SYSTEM ServerTest
  APPLICATION ServerTestApp
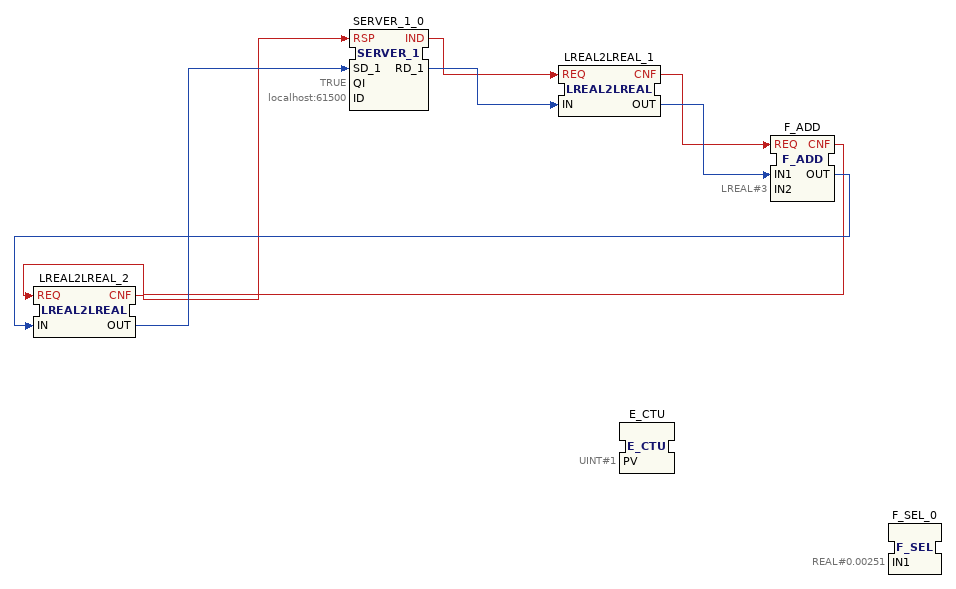
    FBS
      F_ADD : F_ADD(IN2 := LREAL#3);
      SERVER_1_0 : SERVER_1(QI := TRUE, ID := localhost:61500);
      LREAL2LREAL_1 : LREAL2LREAL;
      LREAL2LREAL_2 : LREAL2LREAL;
      E_CTU : E_CTU(PV := UINT#1);
      F_SEL_0 : F_SEL(IN1 := REAL#0.00251);
    END_FBS
    EVENT_CONNECTIONS
      SERVER_1_0.IND TO LREAL2LREAL_1.REQ;
      LREAL2LREAL_1.CNF TO F_ADD.REQ;
      F_ADD.CNF TO LREAL2LREAL_2.REQ;
      LREAL2LREAL_2.CNF TO SERVER_1_0.RSP;
    END_CONNECTIONS
    DATA_CONNECTIONS
      LREAL2LREAL_1.OUT TO F_ADD.IN1;
      SERVER_1_0.RD_1 TO LREAL2LREAL_1.IN;
      F_ADD.OUT TO LREAL2LREAL_2.IN;
      LREAL2LREAL_2.OUT TO SERVER_1_0.SD_1;
    END_CONNECTIONS
  END_APPLICATION
  APPLICATION ServerTestApp2
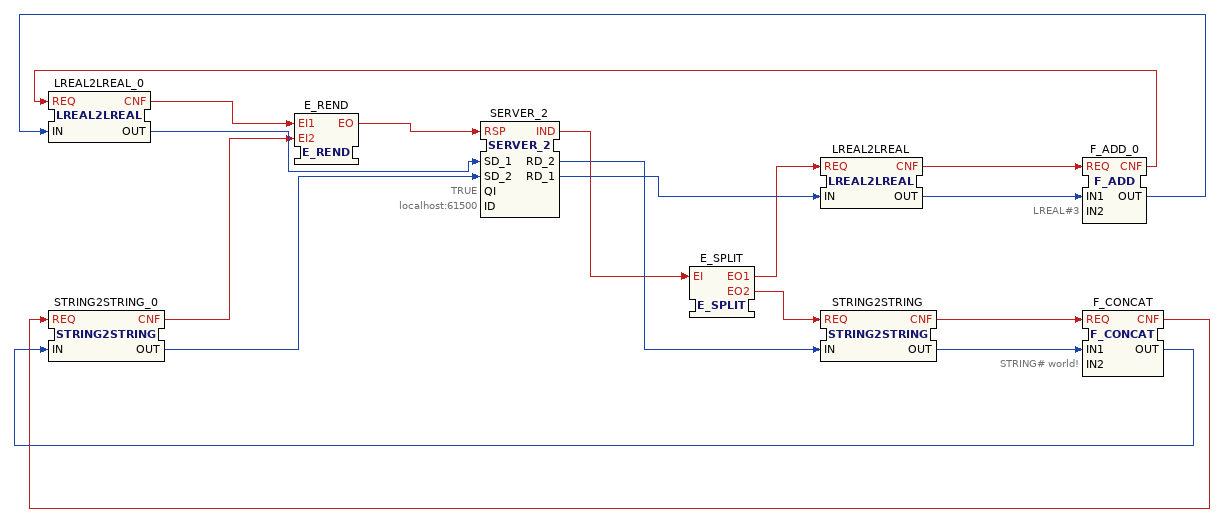
    FBS
      F_ADD_0 : F_ADD(IN2 := LREAL#3);
      F_CONCAT : F_CONCAT(IN2 := STRING# world!);
      SERVER_2 : SERVER_2(QI := TRUE, ID := localhost:61500);
      STRING2STRING : STRING2STRING;
      LREAL2LREAL : LREAL2LREAL;
      E_SPLIT : E_SPLIT;
      E_REND : E_REND;
      STRING2STRING_0 : STRING2STRING;
      LREAL2LREAL_0 : LREAL2LREAL;
    END_FBS
    EVENT_CONNECTIONS
      SERVER_2.IND TO E_SPLIT.EI;
      E_SPLIT.EO1 TO LREAL2LREAL.REQ;
      E_SPLIT.EO2 TO STRING2STRING.REQ;
      LREAL2LREAL.CNF TO F_ADD_0.REQ;
      STRING2STRING.CNF TO F_CONCAT.REQ;
      F_ADD_0.CNF TO LREAL2LREAL_0.REQ;
      F_CONCAT.CNF TO STRING2STRING_0.REQ;
      LREAL2LREAL_0.CNF TO E_REND.EI1;
      STRING2STRING_0.CNF TO E_REND.EI2;
      E_REND.EO TO SERVER_2.RSP;
    END_CONNECTIONS
    DATA_CONNECTIONS
      SERVER_2.RD_2 TO STRING2STRING.IN;
      STRING2STRING.OUT TO F_CONCAT.IN1;
      SERVER_2.RD_1 TO LREAL2LREAL.IN;
      LREAL2LREAL.OUT TO F_ADD_0.IN1;
      F_ADD_0.OUT TO LREAL2LREAL_0.IN;
      F_CONCAT.OUT TO STRING2STRING_0.IN;
      LREAL2LREAL_0.OUT TO SERVER_2.SD_1;
      STRING2STRING_0.OUT TO SERVER_2.SD_2;
    END_CONNECTIONS
  END_APPLICATION
  APPLICATION ServerTestApp3
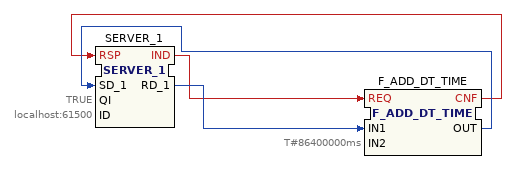
    FBS
      SERVER_1 : SERVER_1(QI := TRUE, ID := localhost:61500);
      F_ADD_DT_TIME : F_ADD_DT_TIME(IN2 := T#86400000ms);
    END_FBS
    EVENT_CONNECTIONS
      SERVER_1.IND TO F_ADD_DT_TIME.REQ;
      F_ADD_DT_TIME.CNF TO SERVER_1.RSP;
    END_CONNECTIONS
    DATA_CONNECTIONS
      SERVER_1.RD_1 TO F_ADD_DT_TIME.IN1;
      F_ADD_DT_TIME.OUT TO SERVER_1.SD_1;
    END_CONNECTIONS
  END_APPLICATION
  APPLICATION ServerTestApp4
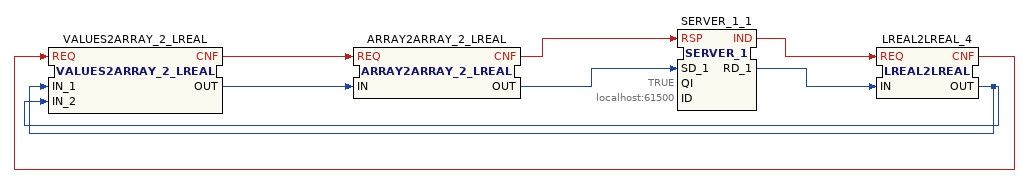
    FBS
      VALUES2ARRAY_2_LREAL : VALUES2ARRAY_2_LREAL;
      SERVER_1_1 : SERVER_1(QI := TRUE, ID := localhost:61500);
      ARRAY2ARRAY_2_LREAL : ARRAY2ARRAY_2_LREAL;
      LREAL2LREAL_4 : LREAL2LREAL;
    END_FBS
    EVENT_CONNECTIONS
      VALUES2ARRAY_2_LREAL.CNF TO ARRAY2ARRAY_2_LREAL.REQ;
      ARRAY2ARRAY_2_LREAL.CNF TO SERVER_1_1.RSP;
      SERVER_1_1.IND TO LREAL2LREAL_4.REQ;
      LREAL2LREAL_4.CNF TO VALUES2ARRAY_2_LREAL.REQ;
    END_CONNECTIONS
    DATA_CONNECTIONS
      VALUES2ARRAY_2_LREAL.OUT TO ARRAY2ARRAY_2_LREAL.IN;
      SERVER_1_1.RD_1 TO LREAL2LREAL_4.IN;
      LREAL2LREAL_4.OUT TO VALUES2ARRAY_2_LREAL.IN_1;
      LREAL2LREAL_4.OUT TO VALUES2ARRAY_2_LREAL.IN_2;
      ARRAY2ARRAY_2_LREAL.OUT TO SERVER_1_1.SD_1;
    END_CONNECTIONS
  END_APPLICATION
  APPLICATION ServerTest5
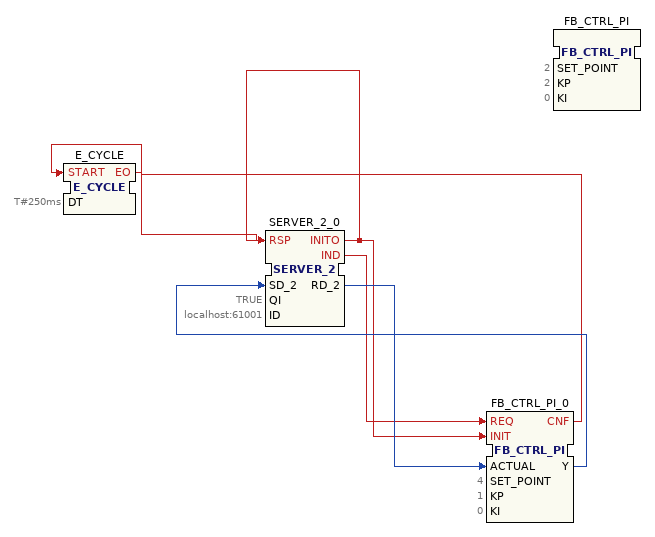
    FBS
      SERVER_2_0 : SERVER_2(QI := TRUE, ID := localhost:61001);
      FB_CTRL_PI : FB_CTRL_PI(SET_POINT := 2, KP := 2, KI := 0);
      FB_CTRL_PI_0 : FB_CTRL_PI(SET_POINT := 4, KP := 1, KI := 0);
      E_CYCLE : E_CYCLE(DT := T#250ms);
    END_FBS
    EVENT_CONNECTIONS
      SERVER_2_0.INITO TO SERVER_2_0.RSP;
      SERVER_2_0.IND TO FB_CTRL_PI_0.REQ;
      SERVER_2_0.INITO TO FB_CTRL_PI_0.INIT;
      FB_CTRL_PI_0.CNF TO E_CYCLE.START;
      E_CYCLE.EO TO SERVER_2_0.RSP;
    END_CONNECTIONS
    DATA_CONNECTIONS
      SERVER_2_0.RD_2 TO FB_CTRL_PI_0.ACTUAL;
      FB_CTRL_PI_0.Y TO SERVER_2_0.SD_2;
    END_CONNECTIONS
  END_APPLICATION
  DEVICE FORTE_PC : FORTE_PC(MGR_ID := "localhost:61499")
    {SET_ATTRIBUTE(Profile, HOLOBLOC)}
    RESOURCE EMB_RES : EMB_RES
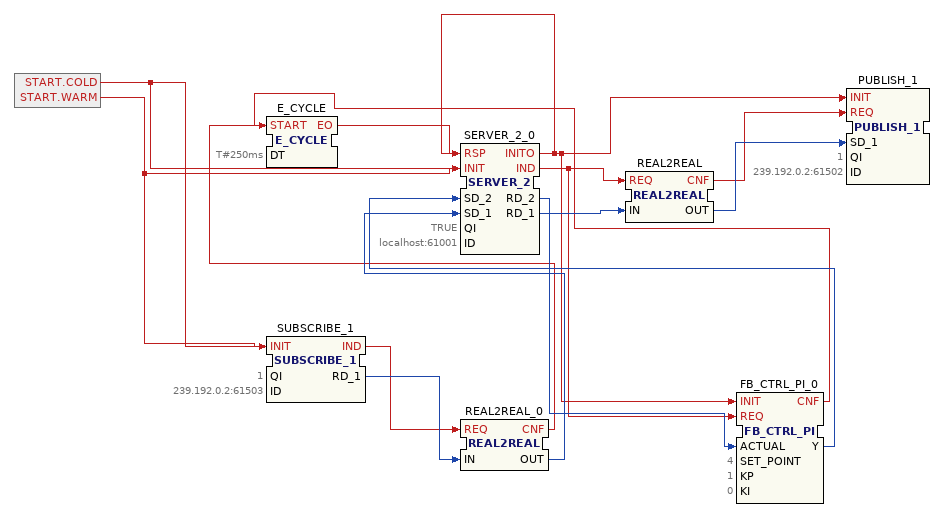
      FBS
        SERVER_2_0 : SERVER_2(QI := TRUE, ID := localhost:61001);
        FB_CTRL_PI_0 : FB_CTRL_PI(SET_POINT := 4, KP := 1, KI := 0);
        E_CYCLE : E_CYCLE(DT := T#250ms);
        REAL2REAL : REAL2REAL;
        PUBLISH_1 : PUBLISH_1(QI := 1, ID := 239.192.0.2:61502);
        SUBSCRIBE_1 : SUBSCRIBE_1(QI := 1, ID := 239.192.0.2:61503);
        REAL2REAL_0 : REAL2REAL;
      END_FBS
      EVENT_CONNECTIONS
        SERVER_2_0.INITO TO SERVER_2_0.RSP;
        SERVER_2_0.INITO TO FB_CTRL_PI_0.INIT;
        SERVER_2_0.IND TO FB_CTRL_PI_0.REQ;
        FB_CTRL_PI_0.CNF TO E_CYCLE.START;
        E_CYCLE.EO TO SERVER_2_0.RSP;
        START.COLD TO SERVER_2_0.INIT;
        START.WARM TO SERVER_2_0.INIT;
        SERVER_2_0.IND TO REAL2REAL.REQ;
        SERVER_2_0.INITO TO PUBLISH_1.INIT;
        REAL2REAL.CNF TO PUBLISH_1.REQ;
        START.COLD TO SUBSCRIBE_1.INIT;
        START.WARM TO SUBSCRIBE_1.INIT;
        SUBSCRIBE_1.IND TO REAL2REAL_0.REQ;
        REAL2REAL_0.CNF TO E_CYCLE.START;
      END_CONNECTIONS
      DATA_CONNECTIONS
        SERVER_2_0.RD_2 TO FB_CTRL_PI_0.ACTUAL;
        FB_CTRL_PI_0.Y TO SERVER_2_0.SD_2;
        SERVER_2_0.RD_1 TO REAL2REAL.IN;
        REAL2REAL.OUT TO PUBLISH_1.SD_1;
        REAL2REAL_0.OUT TO SERVER_2_0.SD_1;
        SUBSCRIBE_1.RD_1 TO REAL2REAL_0.IN;
      END_CONNECTIONS
    END_RESOURCE
  END_DEVICE
  DEVICE FORTE_PC_1 : FORTE_PC(MGR_ID := "localhost:61500")
    {SET_ATTRIBUTE(Profile, HOLOBLOC)}
    RESOURCE EMB_RES : EMB_RES
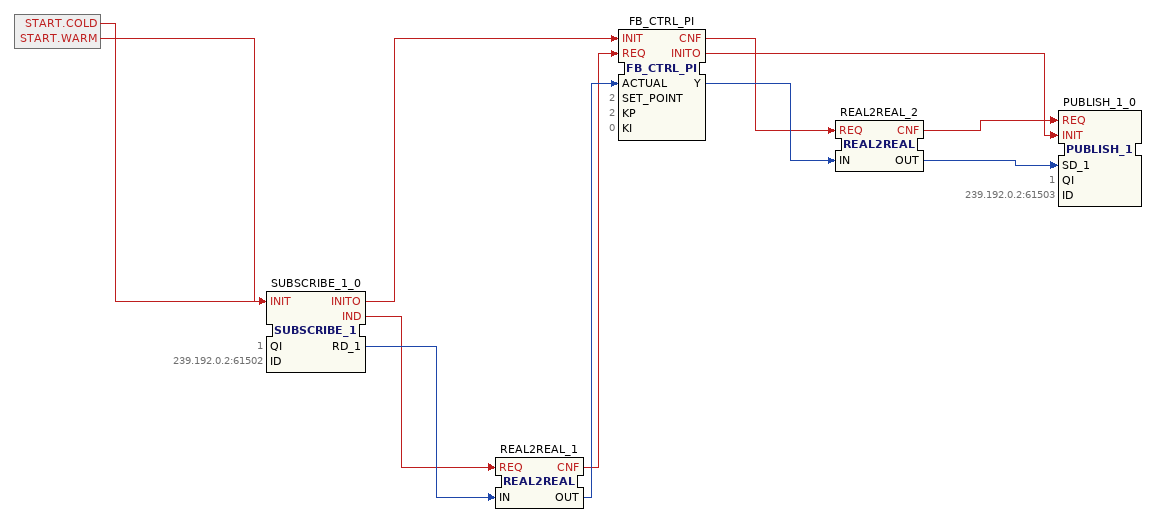
      FBS
        FB_CTRL_PI : FB_CTRL_PI(SET_POINT := 2, KP := 2, KI := 0);
        SUBSCRIBE_1_0 : SUBSCRIBE_1(QI := 1, ID := 239.192.0.2:61502);
        PUBLISH_1_0 : PUBLISH_1(QI := 1, ID := 239.192.0.2:61503);
        REAL2REAL_1 : REAL2REAL;
        REAL2REAL_2 : REAL2REAL;
      END_FBS
      EVENT_CONNECTIONS
        START.COLD TO SUBSCRIBE_1_0.INIT;
        START.WARM TO SUBSCRIBE_1_0.INIT;
        SUBSCRIBE_1_0.INITO TO FB_CTRL_PI.INIT;
        SUBSCRIBE_1_0.IND TO REAL2REAL_1.REQ;
        REAL2REAL_1.CNF TO FB_CTRL_PI.REQ;
        FB_CTRL_PI.CNF TO REAL2REAL_2.REQ;
        REAL2REAL_2.CNF TO PUBLISH_1_0.REQ;
        FB_CTRL_PI.INITO TO PUBLISH_1_0.INIT;
      END_CONNECTIONS
      DATA_CONNECTIONS
        SUBSCRIBE_1_0.RD_1 TO REAL2REAL_1.IN;
        REAL2REAL_1.OUT TO FB_CTRL_PI.ACTUAL;
        FB_CTRL_PI.Y TO REAL2REAL_2.IN;
        REAL2REAL_2.OUT TO PUBLISH_1_0.SD_1;
      END_CONNECTIONS
    END_RESOURCE
  END_DEVICE
  DEVICE FORTE_PC_2 : FORTE_PC(MGR_ID := "localhost:61501")
    {SET_ATTRIBUTE(Profile, HOLOBLOC)}
    RESOURCE EMB_RES : EMB_RES
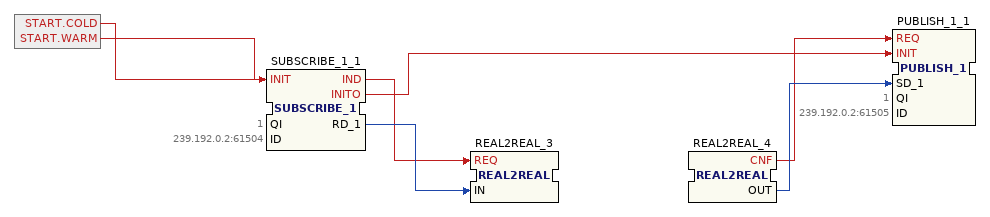
      FBS
        REAL2REAL_3 : REAL2REAL;
        SUBSCRIBE_1_1 : SUBSCRIBE_1(QI := 1, ID := 239.192.0.2:61504);
        PUBLISH_1_1 : PUBLISH_1(QI := 1, ID := 239.192.0.2:61505);
        REAL2REAL_4 : REAL2REAL;
      END_FBS
      EVENT_CONNECTIONS
        START.COLD TO SUBSCRIBE_1_1.INIT;
        START.WARM TO SUBSCRIBE_1_1.INIT;
        SUBSCRIBE_1_1.IND TO REAL2REAL_3.REQ;
        REAL2REAL_4.CNF TO PUBLISH_1_1.REQ;
        SUBSCRIBE_1_1.INITO TO PUBLISH_1_1.INIT;
      END_CONNECTIONS
      DATA_CONNECTIONS
        SUBSCRIBE_1_1.RD_1 TO REAL2REAL_3.IN;
        REAL2REAL_4.OUT TO PUBLISH_1_1.SD_1;
      END_CONNECTIONS
    END_RESOURCE
  END_DEVICE
  MAPPINGS
    ServerTest5.SERVER_2_0 ON FORTE_PC.EMB_RES.SERVER_2_0;
    ServerTest5.FB_CTRL_PI ON FORTE_PC_1.EMB_RES.FB_CTRL_PI;
    ServerTest5.FB_CTRL_PI_0 ON FORTE_PC.EMB_RES.FB_CTRL_PI_0;
    ServerTest5.E_CYCLE ON FORTE_PC.EMB_RES.E_CYCLE;
  END_MAPPINGS
  SEGMENTS
    Ethernet : Ethernet;
  END_SEGMENTS
  LINKS
    FORTE_PC => Ethernet;
    FORTE_PC_1 => Ethernet;
    FORTE_PC_2 => Ethernet;
  END_LINKS
END_SYSTEM
